// TIA Portal project "AB2 Autom Final" (V15)
// Vorlageprojekt für das Buch mit Zielsystem S7-1200

(* hardware
DEVICE "S7-1200-Station_1"  S7-1200 Station
   slot 0: "Baugruppenträger_0"  Rack  V1.0
   slot 1: "PLC_1"  CPU 1211C DC/DC/DC  6ES7 211-1AE40-0XB0  V4.1
*)

// ===== PLC "PLC_1"  CPU 1211C DC/DC/DC =====

VAR_GLOBAL   // PLC tag table "Standard-Variablentabelle"
   "At exit" AT %E0.0 : Bool;
   "Start" AT %E0.1 : Bool;
   "Reset" AT %I0.2 : Bool;
   "Stop" AT %I0.3 : Bool;
   "Emergency stop" AT %I0.4 : Bool;
   "Auto" AT %I0.5 : Bool;
   "FACTORY I/O (Running)" AT %I0.6 : Bool;
   "Vision sensor" AT %ID30 : DInt;
   "Entry conveyor" AT %Q0.0 : Bool;
   "Stop blade" AT %Q0.1 : Bool;
   "Exit conveyor" AT %Q0.2 : Bool;
   "Sorter 1 turn" AT %Q0.3 : Bool;
   "Sorter 1 belt" AT %Q0.4 : Bool;
   "Sorter 2 turn" AT %Q0.5 : Bool;
   "Sorter 2 belt" AT %Q0.6 : Bool;
   "Sorter 3 turn" AT %Q0.7 : Bool;
   "Sorter 3 belt" AT %Q1.0 : Bool;
   "Start light" AT %Q1.1 : Bool;
   "Reset light" AT %Q1.2 : Bool;
   "Stop light" AT %Q1.3 : Bool;
   "Counter 1" AT %QD30 : DInt;
   "Counter 2" AT %QD34 : DInt;
   "Counter 3" AT %QD38 : DInt;
   "Vision sensor in range" AT %M1.0 : Bool;
   "Stop entry conveyor" AT %M1.2 : Bool;
   "Run mode" AT %M1.1 : Bool;
   "Blue range" AT %M1.3 : Bool;
   "Green range" AT %M1.4 : Bool;
   "Blue aux" AT %M1.5 : Bool;
   "Green aux" AT %M1.6 : Bool;
END_VAR

// folder: System blocks/Program resources

DATA_BLOCK "IEC_Timer_0_DB_3"   // DB1
{ S7_Optimized_Access := 'TRUE' }
AUTHOR : Simatic
FAMILY : IEC
NAME : IEC_TMR
VERSION : 1.0
// stored: InstanceOfName IEC_TIMER
"IEC_TIMER"
BEGIN
END_DATA_BLOCK

DATA_BLOCK "Blue counter"   // DB2
{ S7_Optimized_Access := 'TRUE' }
AUTHOR : Simatic
FAMILY : IEC
NAME : CNTR
VERSION : 1.0
// stored: InstanceOfName IEC_COUNTER
"IEC_COUNTER"
BEGIN
END_DATA_BLOCK

DATA_BLOCK "Green counter"   // DB5
{ S7_Optimized_Access := 'TRUE' }
AUTHOR : Simatic
FAMILY : IEC
NAME : CNTR
VERSION : 1.0
// stored: InstanceOfName IEC_COUNTER
"IEC_COUNTER"
BEGIN
END_DATA_BLOCK

DATA_BLOCK "Green delay"   // DB6
{ S7_Optimized_Access := 'TRUE' }
AUTHOR : Simatic
FAMILY : IEC
NAME : IEC_TMR
VERSION : 1.0
// stored: InstanceOfName IEC_TIMER
"IEC_TIMER"
BEGIN
END_DATA_BLOCK

DATA_BLOCK "Blue delay"   // DB7
{ S7_Optimized_Access := 'TRUE' }
AUTHOR : Simatic
FAMILY : IEC
NAME : IEC_TMR
VERSION : 1.0
// stored: InstanceOfName IEC_TIMER
"IEC_TIMER"
BEGIN
END_DATA_BLOCK

// folder: (top level)

FUNCTION "MHJ-PLC-Lab-Function-S71200" : Void   // FC9000, SCL
{ S7_Optimized_Access := 'TRUE' }
VERSION : 0.1
   VAR_TEMP
      rdTimeReturn : Int;
      outputTime : DTL;
      SyncVal : Byte;
      forVal : Int;
      forVal_2 : Int;
      Value : Byte;
   END_VAR
   VAR CONSTANT
      CompVal : Byte := 16#34;
      Value_01 : Byte := 16#11;
      Value_01_DW : DWord := 16#A165_D992;
      Value_02_DW : DWord := 16#58BE_4401;
   END_VAR
BEGIN

   #Value:=PEEK(area := 16#82,
        dbNumber := 0,
        byteOffset := 511);
   #Value := #Value + 1;

   POKE(area := 16#82,
        dbNumber := 0,
        byteOffset := 511,
        value := #Value);

   POKE(area:=16#81,
        dbNumber:=0,
        byteOffset:=1016,
        value:=#Value_01_DW);
   POKE(area := 16#81,
        dbNumber := 0,
        byteOffset := 1020,
        value := #Value_02_DW);

   POKE(area := 16#81,
        dbNumber := 0,
        byteOffset := 511,
        value := B#16#00);

   FOR #forVal := 0 TO 120 DO
       FOR #forVal_2:=0 TO 10 DO
           #rdTimeReturn:=RD_SYS_T(#outputTime);
           #rdTimeReturn := WR_SYS_T(#outputTime);
           #rdTimeReturn := RD_SYS_T(#outputTime);
           #rdTimeReturn := WR_SYS_T(#outputTime);
       END_FOR;
       #SyncVal:= PEEK(area := 16#81,
                      dbNumber := 0,
                      byteOffset := 511);
       IF #SyncVal = #CompVal THEN
          GOTO M_1;
       END_IF;
   END_FOR;
   RETURN;

   M_1:
   POKE(area := 16#81,
        dbNumber := 0,
        byteOffset := 511,
        value := B#16#0);
END_FUNCTION

ORGANIZATION_BLOCK "Main"   // OB1, LAD, ProgramCycle
TITLE = "Main Program Sweep (Cycle)"
{ S7_Optimized_Access := 'TRUE' }
VERSION : 0.1
   VAR_INPUT
      Initial_Call : Bool;   // Initial call of this OB
      Remanence : Bool;   // =True, if remanent data are available
   END_VAR
BEGIN

REGION Network 1: Konnektierungsbaustein für PLC-Lab
   // Im Netzwerk 1 wird der Konnektierungsbaustein für PLC-Lab aufgerufen.
   // Dieser Aufruf darf nicht entfernt werden!
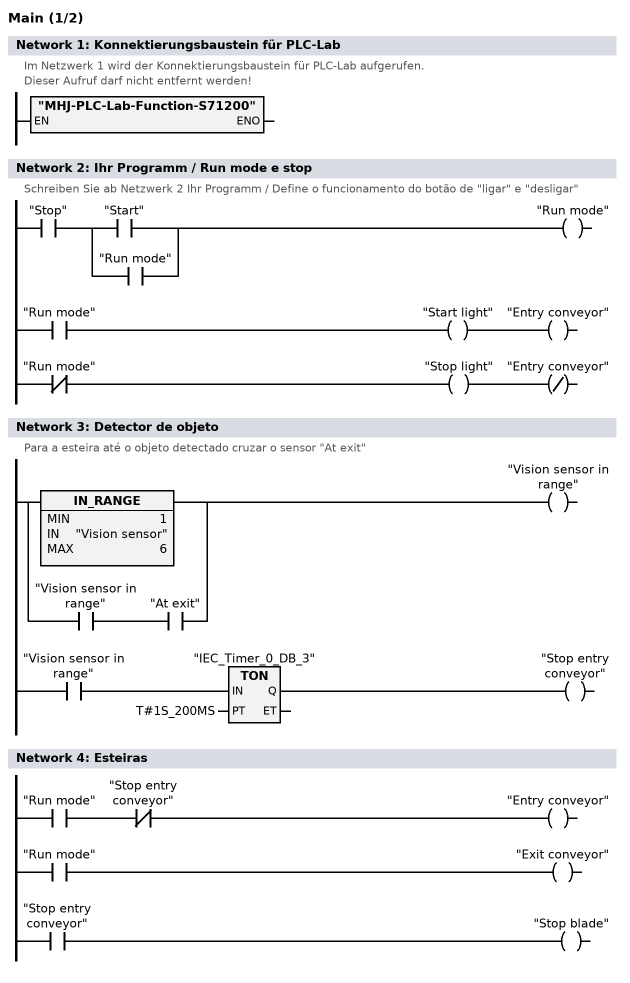
   RUNG wire#powerrail
      "MHJ-PLC-Lab-Function-S71200"()
   END_RUNG
   // the same network as SCL:
   "MHJ-PLC-Lab-Function-S71200"();
END_REGION

REGION Network 2: Ihr Programm / Run mode e stop
   // Schreiben Sie ab Netzwerk 2 Ihr Programm / Define o funcionamento do botão de "ligar" e "desligar"
   RUNG wire#powerrail
      Contact( "Stop" )
      wire#w1
      Contact( "Start" )
      wire#w2
      Coil( "Run mode" )
   END_RUNG
   RUNG wire#w1
      Contact( "Run mode" )
   END_RUNG wire#w2
   RUNG wire#powerrail
      Contact( "Run mode" )
      Coil( "Start light" )
      Coil( "Entry conveyor" )
   END_RUNG
   RUNG wire#powerrail
      I_Contact( "Run mode" )
      Coil( "Stop light" )
      I_Coil( "Entry conveyor" )
   END_RUNG
   // the same network as SCL:
   "Run mode" := "Stop" AND ("Start" OR "Run mode");
   "Start light" := "Run mode";
   "Entry conveyor" := "Run mode";
   "Stop light" := NOT "Run mode";
   "Entry conveyor" := NOT (NOT "Run mode");
END_REGION

REGION Network 3: Detector de objeto
   // Para a esteira até o objeto detectado cruzar o sensor "At exit"
   "Vision sensor in range" := ((1 <= "Vision sensor") AND ("Vision sensor" <= 6)) OR ("Vision sensor in range" AND "At exit");
   "IEC_Timer_0_DB_3".TON(IN := "Vision sensor in range", PT := T#1S_200MS);
   "Stop entry conveyor" := "IEC_Timer_0_DB_3".Q;
END_REGION

REGION Network 4: Esteiras
   RUNG wire#powerrail
      Contact( "Run mode" )
      I_Contact( "Stop entry conveyor" )
      Coil( "Entry conveyor" )
   END_RUNG
   RUNG wire#powerrail
      Contact( "Run mode" )
      Coil( "Exit conveyor" )
   END_RUNG
   RUNG wire#powerrail
      Contact( "Stop entry conveyor" )
      Coil( "Stop blade" )
   END_RUNG
   // the same network as SCL:
   "Entry conveyor" := "Run mode" AND NOT "Stop entry conveyor";
   "Exit conveyor" := "Run mode";
   "Stop blade" := "Stop entry conveyor";
END_REGION

REGION Network 5: Detector de azul
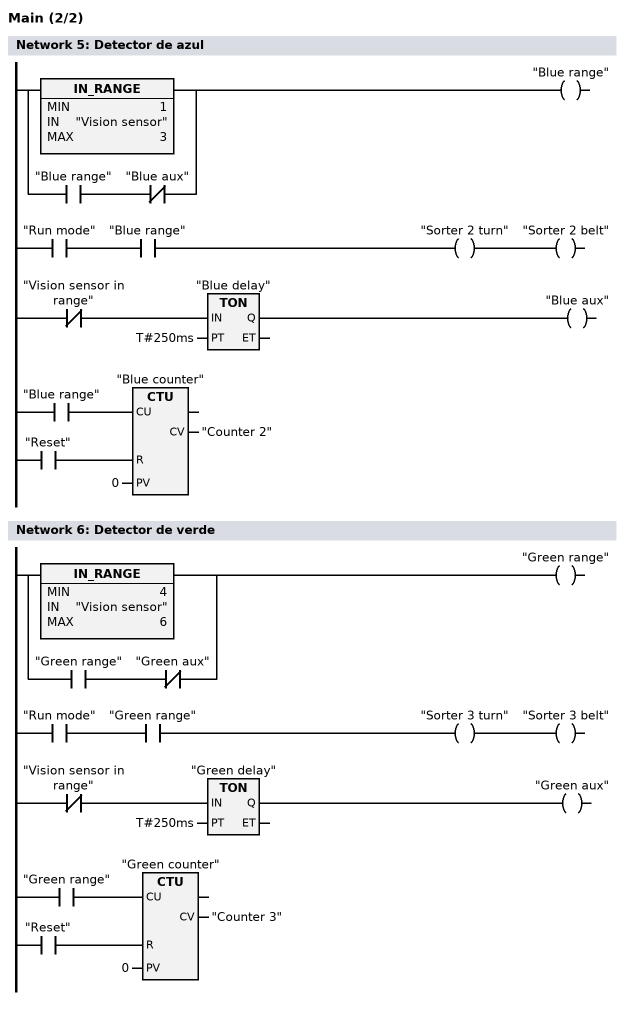
   "Blue range" := ((1 <= "Vision sensor") AND ("Vision sensor" <= 3)) OR ("Blue range" AND NOT "Blue aux");
   "Sorter 2 turn" := "Run mode" AND "Blue range";
   "Sorter 2 belt" := "Sorter 2 turn";
   "Blue delay".TON(IN := NOT "Vision sensor in range", PT := T#250ms);
   "Blue aux" := "Blue delay".Q;
   "Blue counter".CTU(CU := "Blue range", R := "Reset", PV := 0, CV => "Counter 2");
END_REGION

REGION Network 6: Detector de verde
   "Green range" := ((4 <= "Vision sensor") AND ("Vision sensor" <= 6)) OR ("Green range" AND NOT "Green aux");
   "Sorter 3 turn" := "Run mode" AND "Green range";
   "Sorter 3 belt" := "Sorter 3 turn";
   "Green delay".TON(IN := NOT "Vision sensor in range", PT := T#250ms);
   "Green aux" := "Green delay".Q;
   "Green counter".CTU(CU := "Green range", R := "Reset", PV := 0, CV => "Counter 3");
END_REGION
END_ORGANIZATION_BLOCK